FUNCTION_BLOCK FB_Warehouse
VAR_INPUT
END_VAR
VAR_OUTPUT
    nSumme : UINT;
    fMittelwert : REAL;
    nMinWert : UINT;
    nMaxWert : UINT;
END_VAR
VAR
    aStorage : ARRAY[1..7,1..12] OF UINT;
    // Current column
    iX : INT := 1;
    // Current row
    iY : INT := 1;

    iLastStoredMaterial : UINT;
    iLastUnloadedMaterial : UINT;
END_VAR

METHOD PRIVATE RefreshStatistics : BOOL
VAR_INPUT
    nMaterialCount : INT := 0;
END_VAR
// Set all statistics to 0
nSumme := 0;
fMittelwert := 0;
nMinWert := 65535;
nMaxWert := 0;

WHILE iY <= 7 DO
    WHILE iX <= 12 DO
        IF aStorage[iY, iX] <> 0 THEN
            // Increase temporary counter for average calculation
            nMaterialCount := nMaterialCount + 1;

            // Calculate sum of material numbers
            nSumme := nSumme + aStorage[iY, iX];

            // Get lowest material number
            IF nMinWert > aStorage[iY, iX] THEN
                nMinWert := aStorage[iY, iX];
            END_IF

            // Get highest material number
            IF nMaxWert < aStorage[iY, iX] THEN
                nMaxWert := aStorage[iY, iX];
            END_IF
        END_IF

        iX := iX + 1;
    END_WHILE

    iY := iY + 1;
END_WHILE

// Calculate average
END_METHOD

METHOD Store : BOOL
VAR_INPUT
    iMaterialNumber : UINT;
END_VAR
IF iMaterialNumber = 0 THEN
    Store := FALSE;
    RETURN;
END_IF

// Prevent multiple input of same material number
IF iMaterialNumber = iLastStoredMaterial THEN
    Store := FALSE;
    RETURN;
ELSE
    iLastStoredMaterial := iMaterialNumber;
    iX := 1;
    iY := 1;
END_IF

WHILE iY <= 7 DO
    WHILE iX <= 12 DO
        IF aStorage[iY, iX] = 0 THEN
            aStorage[iY, iX] := iMaterialNumber;
            Store := TRUE;
            RETURN;
        END_IF

        iX := iX + 1;
    END_WHILE

    iY := iY + 1;
END_WHILE
END_METHOD

METHOD Unload : BOOL
VAR_INPUT
    iMaterialNumber : UINT;
END_VAR
IF iMaterialNumber = 0 THEN
    Unload := FALSE;
    RETURN;
END_IF

// Prevent multiple input of same material number
IF iMaterialNumber = iLastUnloadedMaterial THEN
    Unload := FALSE;
    RETURN;
ELSE
    iLastUnloadedMaterial := iMaterialNumber;
    iX := 1;
    iY := 1;
END_IF

WHILE iY <= 7 DO
    WHILE iX <= 12 DO
        IF aStorage[iY, iX] = iMaterialNumber THEN
            aStorage[iY, iX] := 0;
            Unload := TRUE;
            RETURN;
        END_IF

        iX := iX + 1;
    END_WHILE

    iY := iY + 1;
END_WHILE
END_METHOD

END_FUNCTION_BLOCK

(* stored: Version 1.1.0.1
   POU FB_Warehouse: Id {6b75effa-3e16-42b7-b2f7-a7912269ea40}, SpecialFunc None
   Method RefreshStatistics: Id {d17ab08b-5503-45ad-8289-e777bacfd648}
   Method Store: Id {a4774fbb-a7d3-4e50-96fa-61783185cd1a}
   Method Unload: Id {b94e3581-2b6f-47be-979a-603286804c4f} *)
